TYPE UDT_CriticalProcessParameters_JacketStripping_RD :
STRUCT
  
  blowTime :UDINT;
  firstCutTime :UDINT;
  firstOpenTime :UDINT;
  SecondCutTime :UDINT;
  secondOpenTime:UDINT;
  secondCutEnable	:BOOL;
  thirdCutTime	:UDINT;
  thirdOpenTime	:UDINT;
  thirdCutEnable	:BOOL;
  fourthCutTime	:UDINT;
  fourthOpenTime:	UDINT;
  fourthCutEnable	:BOOL;
  fifthCutTime	:UDINT;
  fifthOpenTime	:UDINT;
  fifthCutEnable	:BOOL;
  override :INT;
  
END_STRUCT
END_TYPE

(* stored: Version 1.1.0.1, ProductVersion 3.1.4024.12
   DUT UDT_CriticalProcessParameters_JacketStripping_RD: Id {f377f830-cc04-4f50-8a0f-25734a85cac8} *)
